FUNCTION_BLOCK FB_RW_Ctrl EXTENDS CycleHandleFB
VAR_INPUT
	Ctrl_ref:			REFERENCE TO Ctrl_Typ;
END_VAR
VAR_OUTPUT
END_VAR
VAR
	MethInitDone:		BOOL;
END_VAR

VAR CONSTANT
// States are global
		
	RW_INIT:						INT:=0;
	RW_RUN:						INT:=10;
	RW_DONE:			INT:=100;
END_VAR

	IF NOT MethInitDone THEN
		MethInitDone	:= Meth_Init();
	END_IF
	
	IF  THIS^.CMD.Pause = FALSE THEN
		
		//-----------------------------
		//State Machine
		//-----------------------------
		CASE THIS^.StepNo OF
			RW_INIT:
				IF THIS^.StepOneShotTrig THEN
					THIS^.Monitoring.StepMessage	:= 'Init: Start.';
					THIS^.Delay(IN:=FALSE);
				ELSIF Meth_Enable(TRUE) THEN
					THIS^.StepNo	:= 	RW_RUN;
				END_IF	
			
			RW_RUN:
				IF THIS^.StepOneShotTrig THEN
					THIS^.Monitoring.StepMessage	:= 'RW Run.';
					THIS^.Delay(IN:=FALSE);
					Meth_Run_OpenLoop(FALSE);
				ELSIF Meth_Run_OpenLoop(TRUE) THEN
					THIS^.StepNo	:= 	RW_DONE;
				END_IF					
				

			RW_DONE:
				IF THIS^.StepOneShotTrig THEN
					THIS^.Monitoring.StepMessage	:= 'RW cycle Done';
				ELSIF Meth_Done(TRUE) THEN
					THIS^.StepNo	:= 	RW_INIT;
				END_IF		
	
		END_CASE
	
	ELSE
		THIS^.Monitoring.StepMessage:= 'Pause';
		
		IF THIS^.Status.Fault = TRUE THEN
		//IF Meth_EmStop(TRUE) THEN
				THIS^.CMD.ResetCycle	:= TRUE;		// Reset the all state machine to start point
		//END_IF
			
		END_IF
		
	END_IF
	
	THIS^.Delay();
	THIS^.CH_Logic();
	
	// Reset Meth_EmStop when at Init State
	IF THIS^.Pause = FALSE THEN
		//Meth_EmStop(FALSE);
	END_IF

METHOD PRIVATE Meth_Done : BOOL
VAR_INPUT
	Execute: 	BOOL;
END_VAR


	//THIS^.Monitoring.StepMessage			:= 'Press 1 engage';
	//THIS^.Monitoring.Error_Text				:= 'Press 1 engage Fail';
	//THIS^.CMD.Deacivate_Sequence_Time_Out	:= TRUE;	// Disable time out to the all sequence
	//THIS^.CMD.DeactivateStepTimeOut			:= TRUE;	// Disable time out to the actual step
	//THIS^.Parameter.TimeOut					:= T#5S;

	THIS^.Status.Done		:= TRUE;
	THIS^.Status.Running	:= FALSE;									
	Meth_Done	:= TRUE;
END_METHOD

METHOD PRIVATE Meth_Enable : BOOL
VAR_INPUT
	Execute: 	BOOL;
END_VAR


IF THIS^.CMD.Start THEN
	
	THIS^.Monitoring.StepMessage			:= 'Start';
	THIS^.Monitoring.Error_Text				:= 'Start Fail';
	THIS^.CMD.Deacivate_Sequence_Time_Out	:= TRUE;	// Disable time out to the all sequence
	THIS^.CMD.DeactivateStepTimeOut			:= TRUE;	// Disable time out to the actual step
	THIS^.Parameter.TimeOut					:= T#0.5S;

	THIS^.CMD.Start			:= FALSE;
	THIS^.Status.Done		:= FALSE;
	THIS^.Status.Running	:= TRUE;
	
	// Reset Commands and Statuses												
	
	Meth_Enable	:= TRUE;
END_IF
END_METHOD

METHOD Meth_Init :BOOL
VAR_INPUT
END_VAR
//resets
Ctrl_ref.IO.EncoderRW.Ctrl.SetCounterCmd:=FALSE;
RwInverter.ctrl.Start:=FALSE;
RwInverter.ctrl.SetVelocity:=0;

Meth_Init:=TRUE;
END_METHOD

METHOD Meth_Rest_IO 
VAR_INPUT
	
END_VAR

RwInverter.ctrl.Start := FALSE;
RwInverter.ctrl.SetVelocity := 0;
END_METHOD

METHOD Meth_Run_OpenLoop : BOOL
VAR_INPUT
	Excute:BOOL;
END_VAR

IF Excute = FALSE THEN
	THIS^.SubStepNo :=0;
ELSIF Excute AND_THEN THIS^.SubStepNo = 0 THEN
	THIS^.SubStepNo :=10;
END_IF


CASE THIS^.SubStepNo OF
	
	0://Wait
		THIS^.Monitoring.SubStepMessage	:= 'Wait';
		Ctrl_ref.IO.EncoderRW.Ctrl.SetCounterCmd:=FALSE;
		
	
	10://Set counter	
		THIS^.Monitoring.SubStepMessage	:= 'Set counter';
		Ctrl_ref.IO.EncoderRW.Ctrl.SetCounterValue:=0;	
		Ctrl_ref.IO.EncoderRW.Ctrl.SetCounterCmd:=TRUE;	
		IF Ctrl_ref.IO.EncoderRW.Status.SetCounterDone
		OR Ctrl_ref.Simulation 	 THEN
			Ctrl_ref.IO.EncoderRW.Ctrl.SetCounterCmd:=FALSE;
			THIS^.SubStepNo				:=20;
		END_IF	
	
	20: //Start motor
		THIS^.Monitoring.SubStepMessage	:= 'Start Motor';
		RwInverter.ctrl.Start:=TRUE;
		RwInverter.ctrl.SetVelocity:= Ctrl_ref.Parameters.MotorVelocity;	
		THIS^.SubStepNo				:=30;
		
	30://Wait position
		THIS^.Monitoring.SubStepMessage	:= 'Wait position';
		IF Ctrl_ref.IO.EncoderRW.Status.CounterValue >= Ctrl_ref.Parameters.DistanceToMove
		OR Ctrl_ref.Simulation THEN
			RwInverter.ctrl.Start:=FALSE;
			RwInverter.ctrl.SetVelocity:= 0;
			Meth_Run_OpenLoop:=TRUE;
		END_IF
END_CASE
END_METHOD

END_FUNCTION_BLOCK

(* stored: Version 1.1.0.1, ProductVersion 3.1.4024.3
   POU FB_RW_Ctrl: Id {a5ecec96-6bdd-4c97-bccd-89ec0d51e6b5}, SpecialFunc None
   Method Meth_Done: Id {7552bebf-683f-4f61-b274-0af869d06b79}
   Method Meth_Enable: Id {0457fb81-f436-44fd-81cd-fbfa794f7765}
   Method Meth_Init: Id {21c830c1-0a80-405c-991d-f492e5dbb841}
   Method Meth_Rest_IO: Id {d257e215-ad84-45d5-9ddc-cfb2dba58a81}
   Method Meth_Run_OpenLoop: Id {c85cef2f-fa52-415e-80f2-bed9ee0a6aee} *)
